FUNCTION_BLOCK SkillConfig (* Simple FB with one algorithm *)
  (* Standard: 61499-1 *)
  (* Version 1.0, 2024-07-29, AK123700 *)
  PACKAGE DDBImpl;
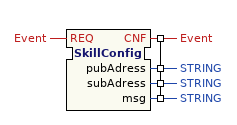
  EVENT_INPUT
    REQ; (* Normal Execution Request *)
  END_EVENT
  EVENT_OUTPUT
    CNF WITH pubAdress, subAdress, msg; (* Execution Confirmation *)
  END_EVENT
  VAR_OUTPUT
    pubAdress : STRING;
    subAdress : STRING;
    msg : STRING;
  END_VAR
  ALGORITHM REQ IN ST:

  END_ALGORITHM
END_FUNCTION_BLOCK
